Staubli VAL3: GoToPos.pgx

public program GoToPos(num x_nAxisNum, num x_nPos)
begin

  if !isPowered()
    popUpMsg("请先给机器人上电")
    return
  endIf
  doStartHoming[x_nAxisNum]=false
  aioSet(aoWorkMode[x_nAxisNum],cst:nPPMODE)
  delay(0.1)
  aioSet(aoPosCmd[x_nAxisNum],x_nPos*nResolution[x_nAxisNum]/nScaleFact[x_nAxisNum])
  delay(0.1)
  doStartHoming[x_nAxisNum]=true
  doManual[x_nAxisNum]=true
  wait(diTargetReach[x_nAxisNum]==false)
  wait(diTargetReach[x_nAxisNum]==true)
  disablePower()
  delay(0.1)
  aioSet(aoWorkMode[x_nAxisNum],cst:nINTERPMODE)
  doStartHoming[x_nAxisNum]=true
end
